// TIA Portal V18 export
DATA_BLOCK "ST10_Stopper_InterfaceDB"   // DB1161
{ S7_Optimized_Access := 'TRUE' }
VERSION : 0.1
// stored: AutoNumber false, DBAccessibleFromOPCUA true, DBAccessibleFromWebserver true, IsOnlyStoredInLoadMemory false, IsRetainMemResEnabled false, IsWriteProtectedInAS false, MemoryReserve 100
   VAR
      aDev { S7_SetPoint := 'True'} : Array[1..5] of "ST_Stopper";
      Command { S7_SetPoint := 'True'} : Array[1..5] of "UDT_Stopper_FB";
   END_VAR
BEGIN
END_DATA_BLOCK
